(* IEC 61131-3 sources: MotionTestBenchMaster/Logical/00_AID/Libraries/Sidel_Libraries/ITC/ETHIP_COM, 5 files *)

(* ---- ETHIP_COM.typ ---- *)
TYPE
	ETHIP_Status_Type :
		(
		ETHIP_DISABLED,
		ETHIP_INITIALIZE_FB,
		ETHIP_INITIAL_PING,
		ETHIP_OPEN,
		ETHIP_RUNNING,
		ETHIP_CLOSE,
		ETHIP_PING,
		ETHIP_WAIT_RESET,
		ETHIP_RECONNECTION
		);
END_TYPE

(* ---- ETHIP_COM.fun ---- *)
(********************************************************************
 * COPYRIGHT --  Sidel S.p.a.
 ********************************************************************
 * Library: ETHIP_COM
 * File: ETHIP_COM.fun
 * Author: Andrea.Cortesi
 * Created: August 26, 2015
 ********************************************************************
 * Functions and function blocks of library ETHIP_COM
 ********************************************************************)

FUNCTION_BLOCK ETHIP_COM
	VAR_INPUT
		Enable : BOOL := FALSE; (*Enable Function Block*)
		IP_Address_Partner : STRING[16] := ' '; (*IP Address Partner*)
		Alive_Bit_From_Partner : BOOL := FALSE; (*Alive Bit From Partner*)
		Reset : BOOL := FALSE; (*Reset Button*)
		TimeOut_Value : UINT := 5000; (*(OPTIONAL) TimeOut Value [ms]. Default value if no setting is 5000 [ms]. Min value accepted 3000 [ms]*)
		Config_DataObject : UDINT := 0; (*Pointer to Data Object Configuration*)
	END_VAR
	VAR_OUTPUT
		Error : BOOL := FALSE; (*Error: TimeOut Connnection or Internal Error (ex: Data Object Not correct) or other function error*)
	END_VAR
	VAR
		PING_Partner : IcmpPing := (0);
		ConnectionAttempt : UINT;
		ETHIP_Init : EIPInit := (0);
		ETHIP_Cyclic : EIPCyclic := (0);
		ETHIP_Exit : EIPExit := (0);
		Handle_Init : UDINT := 0;
		Status : UINT := 0;
		Status_Old : UINT := 0;
		Step_Msg_Active : STRING[255] := ' ';
		Step_Msg_Active_Old : STRING[255] := ' ';
		Msg_Error : STRING[255] := ' ';
		Status_String : STRING[255] := ' ';
		Buffer_Status : ARRAY[0..Buffer_Status_MaxLimit] OF STRING[255] := [41(' ')]; (*Buffer Diagnostic for Status Message*)
		Buffer_Status_Index : USINT := 0;
		Timer_StartComDelay : TON := (0);
		Timer_CommTimeOut : TON := (0);
		Error_Internal : BOOL := FALSE;
		Ping_Ok : BOOL := FALSE;
		ComInit : BOOL := FALSE;
		ComStart : BOOL := FALSE;
		ComExit : BOOL := FALSE;
		zzEdge00000 : BOOL;
		zzEdge00001 : BOOL;
		zzEdge00002 : BOOL;
		zzEdge00003 : BOOL;
	END_VAR
END_FUNCTION_BLOCK

(* ---- ETHIP_COM.st ---- *)
(************************************************************************************************************************)
(* COPYRIGHT -- Sidel S.p.a.                                                                                            *)
(************************************************************************************************************************)
(* Library:				ETHIP_COM																						*)
(* Author:				Andrea.Cortesi																					*)
(* Site:				Sidel - Parma - Product Care IO																	*)
(* Created:				August 26, 2015																					*)
(* Description:			This Library manage a communication based on ethernet IP Protocol between plc B&R configurated	*)
(*						like a SLAVE and another plc configurated like a MASTER. Connection is openinig only if partner	*)
(*						give positive response at comand ping. In case of timeout connection (5000 ms is default value)	*)
(*						the library close connection, try again to ping partner and if there is no answer generate fault*)
(*						communication. Fault is generate also if there is an error inside Data Object configuration.	*)
(* Restriction:			Call in Fast Task at 30 ms or less.Only one connection can be activated because plc B&R in SLAVE*)
(*						Plc B&R can not be SLAVE of two MASTER at same time!!! Is not possible open two connections like*)
(*						SLAVE concurrently on the same IFx eth port. However is possible open two connections like SLAVE*)
(*						Sconcurrently on two different eth port (ex:IF2 and IF3) with two different IP address class	*)
(* Important Note:		This library open/close connection (with memory release) also in case of program download made	*)
(*						in Copy Mode or Overload Mode.For correct management of Overload Mode is necessaary call istance*)
(*						of ETHIP library with Enable at FALSE inside Exit Transiction of function block in which ETHIP	*)
(*						library istance is called.																		*)
(*----------------------------------------------------------------------------------------------------------------------*)
(* Version History:		v.4.00.0 Date 2015-09-12  Andrea.Cortesi														*)
(* Version History:		v.4.00.1 Date 2017-08-20  Roberto.Bonato														*)
(*																														*)
(*----------------------------------------------------------------------------------------------------------------------*)
(* Development Tool:	B&R Automation Studio V3.0.90.27 SP09															*)
(* Compiler GCC:		V2.95.3; V4.1.1; V4.1.2																			*)
(*----------------------------------------------------------------------------------------------------------------------*)
(* Dependencies:		AsEthIP,AsICMP,AsString,Runtime,Standard														*)
(************************************************************************************************************************)

FUNCTION_BLOCK ETHIP_COM
   (* PING Partner before Communication Initialisation *)
	IF (Enable AND NOT(Ping_Ok) AND NOT(Error)) THEN
		PING_Partner.enable		:= TRUE;
		PING_Partner.pHost		:= ADR(IP_Address_Partner);
		PING_Partner.timeout	:= 500;
		PING_Partner();

		Step_Msg_Active      := 'ETHIP PING';
		Status               := PING_Partner.status;
		ETHIP_COM_Error;	(* Call action ETHIP_COM_Error *)

		CASE PING_Partner.status OF
			0:		(* No Error *)
				Ping_Ok	:= TRUE;

			32750,	(* No response sent by station within the specified timeout *)
			32751,	(* The specified IP address (SG4: name also) could not be resolved *)
			32752,	(* Resource problem in system. Could not create new sockets *)
			65535:	(* No Error - Function block still operating, continue calling *)
				Ping_Ok	:= FALSE;
			ELSE	(* Error not management *)
				Ping_Ok	:= FALSE;
		END_CASE
	END_IF

	(* ETHIP Communication Initialisation *)
	IF ComInit THEN	(* If the communication initialisation is requested then... *)
		ETHIP_Init.enable	:= TRUE;				(* Enabled *)
		ETHIP_Init.pconfig	:= Config_DataObject;	(* Name of the "communication configuration" data object *)
		ETHIP_Init();								(* Call of the "EIPInit" function *)

		Handle_Init			:= ETHIP_Init.handle;	(* The handle returned by the EIPInit Function and is reused by the EIPCyclic AND EIPExit functions *)

		Step_Msg_Active		:= 'ETHIP INIT';
		Status				:= ETHIP_Init.status;
		ETHIP_COM_Error;							(* Call action ETHIP_COM_Error *)

		(* ETHIP Status Init *)
		CASE ETHIP_Init.status OF
			0:		(* No Error *)
				ComInit		:= FALSE;		(* Reset the communication init request *)
				ComStart	:= TRUE;		(* Set the communication activation request *)

			32051,	(* Out of memory. The library cannot be executed *)
			32052,	(* Configuration data object error *)
			32053,	(* Illegal input parameters connected to the FBK. *)
			32054:	(* The Ethernet interface doesn't exist or returns an error. Check the #OWNINTERFACE entry in the configuration data object.*)
				ComInit		:= FALSE;		(* Reset the communication init request *)
				ComStart	:= FALSE;		(* Reset the communication activation request *)
				ComExit		:= TRUE;		(* Set the communication exit request *)

			65534:	(* The FBK was called with enable = 0.*)

			65535:	(* No Error - Function block still operating, continue calling *)

			ELSE	(* Error not management *)
				ComInit		:= FALSE;		(* Reset the communication init request *)
				ComStart	:= FALSE;		(* Reset the communication activation request *)
				ComExit		:= FALSE;		(* Reset the communication exit request *)
		END_CASE
	END_IF

	(* ETHIP Communication Cyclic *)
	IF ComStart THEN		(* If communication activation is requested then... *)
		ETHIP_Cyclic.enable	:= TRUE;		(* Enabled *)
		ETHIP_Cyclic.handle	:= Handle_Init;	(* Handle received from the EIPInit function *)
		ETHIP_Cyclic();						(* Call of the "EIPcyclic" function *)

		Step_Msg_Active		:= 'ETHIP CYCLIC';
		Status				:= ETHIP_Cyclic.status;
		ETHIP_COM_Error;					(* Call action ETHIP_COM_Error *)
	END_IF

	(* ETHIP Status Cyclic *)
	CASE ETHIP_Cyclic.status OF
		0:		(* No Error *)

		32051,	(* Out of memory. The library cannot be executed *)
		32052,	(* Configuration data object error *)
		32053,	(* Illegal input parameters connected to the FBK. *)
		32054:	(* The Ethernet interface doesn't exist or returns an error. Check the #OWNINTERFACE entry in the configuration data object.*)
			ComStart	:= FALSE;		(* Reset the communication activation request *)
			ComExit		:= TRUE;		(* Set the communication exit request *)

		65534:	(* The FBK was called with enable = 0.*)

		65535:	(* No Error - Function block still operating, continue calling *)

		ELSE	(* Error not management *)
			ComInit		:= FALSE;	(* Reset the Communication init request *)
			ComStart	:= FALSE;	(* Reset the communication activation request *)
			ComExit		:= FALSE;	(* Reset the communication exit request *)
	END_CASE

	(* Force ETHIP Communication Exit if Enable Not Active *)
	IF (NOT(Enable) AND (ComStart OR ComInit)) THEN
		ComInit		:= FALSE;	(* Reset the communication init request *)
		ComStart	:= FALSE;	(* Reset the communication activation request *)
		ComExit		:= TRUE;	(* Set the communication exit request *)
	END_IF

	(* ETHIP Communication Exit *)
	IF ComExit THEN	(* If communication exit is requested then... *)
		ComInit		:= FALSE;		(* Reset the communication init request *)
		ComStart	:= FALSE;		(* Reset the communication activation request *)

		ETHIP_Exit.enable	:= TRUE;		(* Enabled *)
		ETHIP_Exit.handle	:= Handle_Init;	(* Handle received from the EIPInit function *)
		ETHIP_Exit();						(* Call of the "EIPExit" function *)

		Step_Msg_Active		:= 'ETHIP EXIT';
		Status				:= ETHIP_Exit.status;
		ETHIP_COM_Error;					(* Call action ETHIP_COM_Error *)
	END_IF

	(* ETHIP Status Exit *)
	CASE ETHIP_Exit.status OF
		0:		(* No Error *)

		32051,	(* Out of memory. The library cannot be executed *)
		32052,	(* Configuration data object error *)
		32053,	(* Illegal input parameters connected to the FBK. *)
		32054:	(* The Ethernet interface doesn't exist or returns an error. Check the #OWNINTERFACE entry in the configuration data object.*)
			ComInit		:= FALSE;	(* Reset the communication init request *)
			ComStart	:= FALSE;	(* Reset the communication activation request *)
			ComExit		:= FALSE;	(* Reset the communication exit request *)

		65534:	(* The FBK was called with enable = 0. *)

		65535:	(* No Error - Function block still operating, continue calling *)

		ELSE	(* Error not management *)
			ComInit		:= FALSE;	(* Reset the communication init request *)
			ComStart	:= FALSE;	(* Reset the communication activation request *)
			ComExit		:= FALSE;	(* Reset the communication exit request *)
	END_CASE

	// Check if ETHIP Communication Exit is Ended
	IF (ComExit AND (ETHIP_Exit.status = 0)) THEN
		ComInit		:= FALSE;		(* Reset the communication init request *)
		ComStart	:= FALSE;		(* Reset the communication activation request *)
		ComExit		:= FALSE;		(* Reset the communication exit request *)
	END_IF

	// Check Presence Status Error in ETHIP Init and ETHIP Cyclic
	IF ((ETHIP_Init.status = 0) OR (ETHIP_Init.status = 65335)) AND ((ETHIP_Cyclic.status = 0) OR (ETHIP_Cyclic.status = 65335)) THEN
		Error_Internal	:= FALSE;	(* Reset Error in ETHIP function *)
	ELSE
		IF Ping_Ok THEN
			Error_Internal	:= TRUE;	(* Set Error in ETHIP function *)
		ELSE
			Error_Internal	:= FALSE;	(* Reset Error in ETHIP function *)
		END_IF
	END_IF

	// Set Communication Exit if Ping Not Ok or Fault Communication
	IF (ComStart AND (EDGEPOS(Error) OR EDGENEG(Ping_Ok))) THEN
		IF ConnectionAttempt > 10 THEN
			ComInit		:= FALSE;		(* Reset the communication init request *)
			ComStart	:= FALSE;		(* Reset the communication activation request *)
			ComExit		:= TRUE;		(* Set the communication exit request *)
			ConnectionAttempt := 0;
		ELSE
			ConnectionAttempt	:= ConnectionAttempt + 1;
			Error := FALSE;
		END_IF
	ELSIF (ComStart AND EDGE(Alive_Bit_From_Partner)) THEN
		ConnectionAttempt := 0;
	END_IF

	// Initializatin Communication
	IF (Enable AND NOT(ComInit) AND NOT(ComStart) AND NOT(ComExit) AND Ping_Ok AND NOT(Error)) THEN
		ComInit		:= TRUE;		(* Set the communication init request *)
		ComStart	:= FALSE;		(* Reset the communication activation request *)
		ComExit		:= FALSE;		(* Reset the communication exit request *)
	END_IF

	// Check TimeOut Value
	IF (TimeOut_Value = 0) THEN
		TimeOut_Value	:= 5000;
	ELSIF (TimeOut_Value < 3000) THEN
		TimeOut_Value	:= 3000;
	END_IF

	// Check Alive Bit Receive from Partner
	IF Enable THEN
		Timer_CommTimeOut(
		IN	:= NOT EDGE(Alive_Bit_From_Partner) AND Timer_StartComDelay.Q,
		PT	:= UINT_TO_TIME(TimeOut_Value)
		);

		Timer_StartComDelay(
		IN	:= TRUE,
		PT	:= UINT_TO_TIME(TimeOut_Value)
		);
	ELSE
		Timer_CommTimeOut(
		IN	:= FALSE,
		PT	:= UINT_TO_TIME(TimeOut_Value)
		);

		Timer_StartComDelay(
		IN	:= FALSE,
		PT	:= UINT_TO_TIME(TimeOut_Value)
		);
	END_IF

	// TimeOut Error Communication
	IF ((NOT(Ping_Ok) AND Timer_CommTimeOut.Q) OR Error_Internal) THEN
		Timer_CommTimeOut.IN	:= FALSE;
		Timer_StartComDelay.IN	:= FALSE;
		Error					:= TRUE;
	END_IF

	// Try again to Ping Partner in case of TimeOut Error Communication
	IF (Ping_Ok AND Timer_CommTimeOut.Q AND NOT(Error)) THEN
		Timer_CommTimeOut.IN	:= FALSE;
		Timer_StartComDelay.IN	:= FALSE;
		Ping_Ok					:= FALSE;
	END_IF

	// Re-initial Communication in CASE OF ERROR
	IF Error THEN
		IF Reset THEN
			Timer_CommTimeOut.IN	:= FALSE;
			Timer_StartComDelay.IN	:= FALSE;
			Error					:= FALSE;
			Ping_Ok					:= FALSE;

			// Reset Buffer and Status
			Buffer_Status_Index		:= 0;
			Status_Old				:= 0;
			Step_Msg_Active_Old		:= '';
			Status_String			:= '';
			memset(ADR(Buffer_Status), 0, SIZEOF(Buffer_Status));

			Step_Msg_Active			:= 'ETHIP RESET';
			Status					:= 55150;	(* Reset Allarm Communication Library *)
			ETHIP_COM_Error;					(* Call action ETHIP_COM_Error *)
		END_IF
	END_IF

	// Call timer
	Timer_CommTimeOut();
	Timer_StartComDelay();
END_FUNCTION_BLOCK

(* ---- ETHIP_COM.var ---- *)
(********************************************************************
 * COPYRIGHT --  Sidel S.p.a
 ********************************************************************
 * Library: ETHIP_COM
 * File: ETHIP_COM.var
 * Author: Andrea.Cortesi
 * Created: August 26, 2015
 ********************************************************************
 * Constants of library ETHIP_COM
 ********************************************************************)
VAR CONSTANT
	Buffer_Status_MaxLimit : USINT := 40;
END_VAR

(* ---- ETHIP_COM_Error.st ---- *)
(********************************************************************
 * COPYRIGHT --  Sidel S.p.a.
 ********************************************************************
 * Program: ETHIP_COM
 * File: ETHIP_COM_Error.st
 * Author: Andrea.Cortesi
 * Created: August 26, 2015
 ********************************************************************
 * Implementation of program ETHIP_COM
 ********************************************************************)

ACTION ETHIP_COM_Error:

	CASE Status OF

		0    : Msg_Error := 'No Error';
		55100: Msg_Error := 'Error Enable Library File_CSV Not Coerent';
		55101: Msg_Error := 'Error File CSV Actual is Empty (size zero)';
		55102: Msg_Error := 'Error File CSV Old is Empty (size zero)';
		55103: Msg_Error := 'Force Exit from Sequencer Library FILE_CSV';
		55104: Msg_Error := 'File CSV Saved - No Error';
		55105: Msg_Error := 'File CSV Loaded - No Error';
		55106: Msg_Error := 'Error Step Sequencer in Library FILE_CSV';
		55150: Msg_Error := 'Reset Error Communication Library';
		9999 : Msg_Error := 'FUNCTION NOT implemented';
		20700: Msg_Error := 'Invalid path; check the path specification (AND length OF path)';
		20701: Msg_Error := 'The specified data length is too small';
		20702: Msg_Error := 'No more file handles available';
		20703: Msg_Error := 'Code error (system error)';
		20704: Msg_Error := 'Invalid TYPE';
		20705: Msg_Error := 'File already exists';
		20706: Msg_Error := 'ACCESS NOT possible using the desired mode';
		20707: Msg_Error := 'FiERR_MODE  Illegal mode';
		20708: Msg_Error := 'File does NOT exist';
		20709: Msg_Error := 'Illegal file device (e.g. not initialized "CPU -> Properties -> File Devices")';
		20710: Msg_Error := 'NOT enough memory FOR file with new write data';
		20711: Msg_Error := 'Invalid file offset';
		20712: Msg_Error := 'File NOT allowed';
		20713: Msg_Error := 'NOT enough memory (DRAM) available TO copy file';
		20714: Msg_Error := 'General error in FileOpen';
		20715: Msg_Error := 'General error in FileClose';
		20716: Msg_Error := 'General error in FileRead';
		20717: Msg_Error := 'General error in FileWrite';
		20718: Msg_Error := 'General error in Ioctl';
		20719: Msg_Error := 'The specified POINTER is invalid (NULL)';
		20720: Msg_Error := 'Error in the FileIO manager';
		20721: Msg_Error := 'File NOT open';
		20722: Msg_Error := 'Invalid directory';
		20723: Msg_Error := 'Directory does NOT exist';
		20724: Msg_Error := 'Directory NOT empty';
		20725: Msg_Error := 'Directory already exists';
		20726: Msg_Error := 'Error retrieving memory information';
		20727: Msg_Error := 'NOT enough memory available on the target device (FileCopy)';
		20728: Msg_Error := 'Idents directory no longer available. Close open directories (or free up memory)';
		20729: Msg_Error := 'Invalid parameter output';
		20730: Msg_Error := 'Directory already exists';
		20731: Msg_Error := 'The specified handle is invalid';
		20732: Msg_Error := 'Another IP address has already been defined FOR a host name';
		20796: Msg_Error := 'Could NOT initialize library';
		20797: Msg_Error := 'Error in device driver';
		20798: Msg_Error := 'Error in device manager';
		20799: Msg_Error := 'System error.General system fault';
		32051: Msg_Error := 'Out of memory. The library cannot be executed';
		32052: Msg_Error := 'Configuration data object error';
		32053: Msg_Error := 'Illegal input parameters connected to the Function block';
		32054: Msg_Error := 'Ethernet interface not exist or in error.Check #OWNINTERFACE data object';
		32750: Msg_Error := 'No response sent by station within the specified timeout';
		32751: Msg_Error := 'The specified IP address (SG4: name also) could not be resolved';
		32752: Msg_Error := 'Resource problem in system. Could not create new sockets';
		32799: Msg_Error := 'System error';
		65534: Msg_Error := 'Function block was called with enable at FALSE';
		65535: Msg_Error := 'Function block continue calling';

	ELSE

			   Msg_Error := 'Error not management';

	END_CASE

	// Buffer Status for Diagnostic
	IF ((Status <> Status_Old) OR ((strcmp(ADR(Step_Msg_Active),ADR(Step_Msg_Active_Old))) <> 0)) AND (Buffer_Status_Index < Buffer_Status_MaxLimit) THEN
		itoa(UINT_TO_DINT(Status),ADR(Status_String));
		Status_String                      := CONCAT(Status_String,': ');
		Status_String                      := CONCAT(Status_String,Step_Msg_Active);
		Status_String                      := CONCAT(Status_String,': ');
		Buffer_Status[Buffer_Status_Index] := CONCAT(Status_String,Msg_Error);
		Buffer_Status_Index                := (Buffer_Status_Index + 1);

		// Update Status Old if Change
		IF (Status <> Status_Old) THEN
			Status_Old := Status;
		END_IF
		// Update Step Msg active Old if Changed
		IF ((strcmp(ADR(Step_Msg_Active),ADR(Step_Msg_Active_Old))) <> 0) THEN
		    Step_Msg_Active_Old := Step_Msg_Active;
		END_IF
		// Reset Buffer Status if is Fu
		IF (Buffer_Status_Index = Buffer_Status_MaxLimit) THEN
		    // Reset Buffer and Status
		    Buffer_Status_Index      := 0;
			Status_Old               := 0;
			Step_Msg_Active_Old      := '';
		    memset(ADR(Buffer_Status),0,SIZEOF(Buffer_Status));
		END_IF

	END_IF

END_ACTION
